(* CoDeSys 2.3.9.50 project: dc-motor.pro *)
(* Libraries: STANDARD.LIB 5.6.98 12:03:02 *)

(* Task configuration *)
TASK Standard (PRIORITY := 0, INTERVAL := T#10ms);
	MAIN
END_TASK

(* POU MAIN, ST *)
PROGRAM MAIN
VAR
END_VAR
;
END_PROGRAM
